(****************************************************************************************)
(*							Beckhoff Automation Poland									*)
(*								FB_AiRMixer  v1											*)
(*									27.05.2008											*)
(*							Bloczek do mieszania powietrza								*)
(*______________________________________________________________________________________*)
FUNCTION_BLOCK FB_AirMixer
VAR_INPUT
	Set:			REAL;
	Tin:			REAL;
	Tout:			REAL:=1;
	UpperLimit:		REAL;
	LowerLimit:		REAL;
END_VAR
VAR_OUTPUT
	Y:				REAL;
	Cool:			BOOL;
	Heat:			BOOL;
END_VAR
VAR
	deltaT:			REAL;
	a:				REAL;
	b:				REAL;
	Wyjscie: 		REAL;
	deltaLimit: 	REAL;
END_VAR

deltaT:=Tout-Tin;
deltaLimit:=UpperLimit-LowerLimit;
(*a:=deltaLimit/deltaT;*)
(*b:=(-deltaLimit*Tin)/deltaT;*)
Wyjscie:=a*Set+b;
IF Wyjscie < LowerLimit THEN
	Y:= LowerLimit;
	Cool:=TRUE;
ELSE Y:=Wyjscie;
END_IF
IF Wyjscie >UpperLimit THEN
	 Y:= UpperLimit;
	Heat:=TRUE;
ELSE Y:= Wyjscie;
END_IF
IF cool = TRUE AND Wyjscie>(LowerLimit+0.2*deltaLimit) THEN cool:=FALSE; END_IF
IF heat = TRUE AND Wyjscie>(UpperLimit-0.2*deltaLimit) THEN heat:=FALSE; END_IF

END_FUNCTION_BLOCK

(* stored: Version 1.1.0.1, ProductVersion 3.1.4019.2
   POU FB_AirMixer: Id {88a7f0fc-d117-492a-88d5-29210a445fac}, SpecialFunc None *)
